% RSLogix 500 project LANE SORT_BAK008.RSS, saved by version 8.30.00.16 %
PROJECT "UNTITLED"    % processor: Bul.1763 MicroLogix 1100 Series B %

PROGRAM FILES
  LAD 2 "MAIN"  2 rungs
  LAD 3 "MTCONTROL"  5 rungs
  LAD 4 "BOX DETECT"  7 rungs

DATA FILES
  O0 OUTPUT  5 elements
  I1 INPUT  7 elements
  S2 STATUS  66 elements
  B3 BINARY  1 elements
  T4 TIMER  2 elements
  C5 COUNTER  2 elements
  R6 CONTROL  1 elements
  N7 INTEGER  10 elements
  F8 FLOAT  1 elements
  N10 SERIAL_NUM  10 elements
  N11 LABELDATA  10 elements
  N12 LABELPRINT  10 elements

LADDER 2 "MAIN"
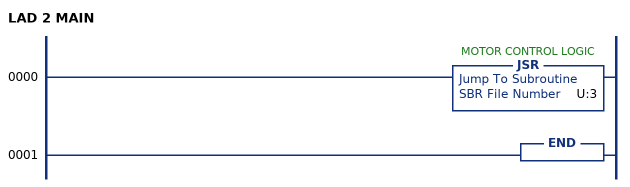
% Rung: 0 %
SOR JSR U:3 EOR
%   U:3  "MOTOR CONTROL LOGIC" %
% Rung: 1 %
SOR END EOR

LADDER 3 "MTCONTROL"
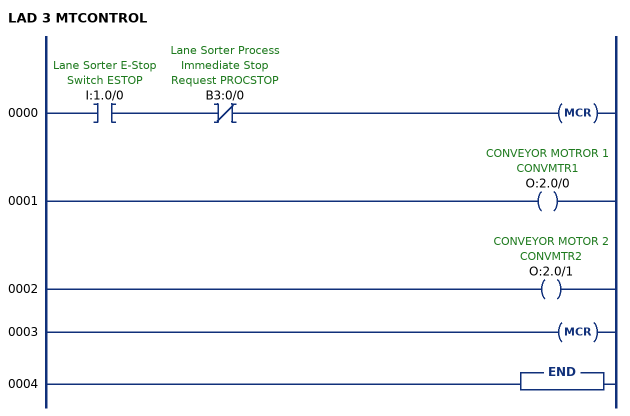
% Rung: 0 %
SOR XIC I:1.0/0 XIO B3:0/0 MCR EOR
%   I:1.0/0  ESTOP  "Lane Sorter E-Stop Switch" %
%   B3:0/0  PROCSTOP  "Lane Sorter Process Immediate Stop Request" %
% Rung: 1 %
SOR OTE O:2.0/0 EOR
%   O:2.0/0  CONVMTR1  "CONVEYOR MOTROR 1" %
% Rung: 2 %
SOR OTE O:2.0/1 EOR
%   O:2.0/1  CONVMTR2  "CONVEYOR MOTOR 2" %
% Rung: 3 %
SOR MCR EOR
% Rung: 4 %
SOR END EOR

LADDER 4 "BOX DETECT"
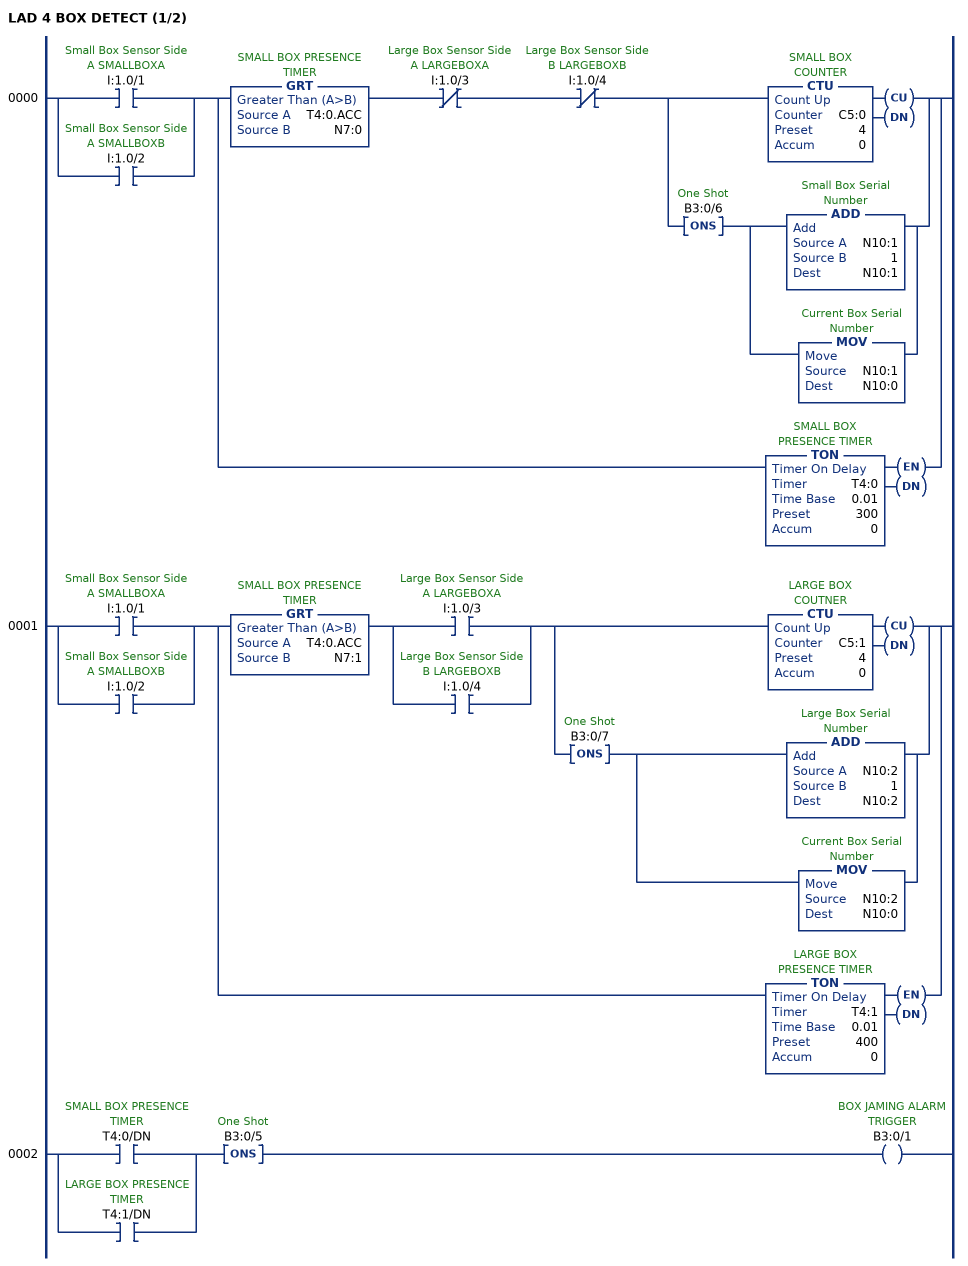
% Rung: 0 %
SOR BST XIC I:1.0/1 NXB XIC I:1.0/2 BND BST GRT T4:0.ACC N7:0 XIO I:1.0/3 XIO I:1.0/4 BST CTU C5:0 4 0 NXB ONS B3:0/6 BST ADD N10:1 1 N10:1 NXB MOV N10:1 N10:0 BND BND NXB TON T4:0 0.01 300 0 BND EOR
%   I:1.0/1  SMALLBOXA  "Small Box Sensor Side A" %
%   I:1.0/2  SMALLBOXB  "Small Box Sensor Side A" %
%   T4:0  "SMALL BOX PRESENCE TIMER" %
%   N7:0  "SMALL BOX DETECTION TIME (ms)" %
%   I:1.0/3  LARGEBOXA  "Large Box Sensor Side A" %
%   I:1.0/4  LARGEBOXB  "Large Box Sensor Side B" %
%   C5:0  "SMALL BOX COUNTER" %
%   B3:0/6  "One Shot" %
%   N10:1  "Small Box Serial Number" %
%   N10:0  "Current Box Serial Number" %
% Rung: 1 %
SOR BST XIC I:1.0/1 NXB XIC I:1.0/2 BND BST GRT T4:0.ACC N7:1 BST XIC I:1.0/3 NXB XIC I:1.0/4 BND BST CTU C5:1 4 0 NXB ONS B3:0/7 BST ADD N10:2 1 N10:2 NXB MOV N10:2 N10:0 BND BND NXB TON T4:1 0.01 400 0 BND EOR
%   I:1.0/1  SMALLBOXA  "Small Box Sensor Side A" %
%   I:1.0/2  SMALLBOXB  "Small Box Sensor Side A" %
%   T4:0  "SMALL BOX PRESENCE TIMER" %
%   N7:1  "LARGE BOX DETECTION TIME (ms)" %
%   I:1.0/3  LARGEBOXA  "Large Box Sensor Side A" %
%   I:1.0/4  LARGEBOXB  "Large Box Sensor Side B" %
%   C5:1  "LARGE BOX COUTNER" %
%   B3:0/7  "One Shot" %
%   N10:2  "Large Box Serial Number" %
%   N10:0  "Current Box Serial Number" %
%   T4:1  "LARGE BOX PRESENCE TIMER" %
% Rung: 2 %
SOR BST XIC T4:0/DN NXB XIC T4:1/DN BND ONS B3:0/5 OTE B3:0/1 EOR
%   T4:0  "SMALL BOX PRESENCE TIMER" %
%   T4:1  "LARGE BOX PRESENCE TIMER" %
%   B3:0/5  "One Shot" %
%   B3:0/1  "BOX JAMING ALARM TRIGGER" %

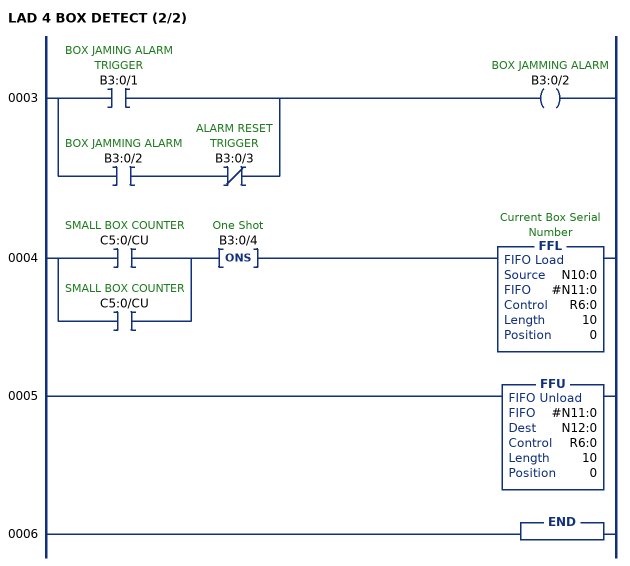
% Rung: 3 %
SOR BST XIC B3:0/1 NXB XIC B3:0/2 XIO B3:0/3 BND OTE B3:0/2 EOR
%   B3:0/1  "BOX JAMING ALARM TRIGGER" %
%   B3:0/2  "BOX JAMMING ALARM" %
%   B3:0/3  "ALARM RESET TRIGGER" %
% Rung: 4 %
SOR BST XIC C5:0/CU NXB XIC C5:0/CU BND ONS B3:0/4 FFL N10:0 #N11:0 R6:0 10 0 EOR
%   C5:0  "SMALL BOX COUNTER" %
%   B3:0/4  "One Shot" %
%   N10:0  "Current Box Serial Number" %
% Rung: 5 %
SOR FFU #N11:0 N12:0 R6:0 10 0 EOR
% Rung: 6 %
SOR END EOR

DATA TABLE (non-zero values as saved)
DATA T4
% .PRE .ACC %
% T4:0 % 300 0
% T4:1 % 400 0
DATA C5
% .PRE .ACC %
% C5:0 % 4 0
% C5:1 % 4 0
DATA R6
% .LEN .POS %
% R6:0 % 10 0
DATA N10
% N10:0 % 0 10000 20000 0 0 0 0 0 0 0
